FUNCTION_BLOCK SIMULATE
  {SET_ATTRIBUTE(OpcUa, SERVICE)}
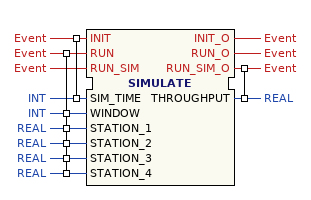
  EVENT_INPUT
    INIT WITH SIM_TIME;
    RUN WITH WINDOW, STATION_1, STATION_2, STATION_3, STATION_4; {SET_ATTRIBUTE(OpcUa, Method)}
    RUN_SIM; {SET_ATTRIBUTE(OpcUa, Method)}
  END_EVENT
  EVENT_OUTPUT
    INIT_O;
    RUN_O;
    RUN_SIM_O WITH THROUGHPUT;
  END_EVENT
  VAR_INPUT
    SIM_TIME : INT; {SET_ATTRIBUTE(OpcUa, Variable.RUN)}
    WINDOW : INT; {SET_ATTRIBUTE(OpcUa, Constant.RUN)}
    STATION_1 : REAL; {SET_ATTRIBUTE(OpcUa, Variable.RUN)}
    STATION_2 : REAL; {SET_ATTRIBUTE(OpcUa, Constant.RUN)}
    STATION_3 : REAL; {SET_ATTRIBUTE(OpcUa, Variable.RUN)}
    STATION_4 : REAL; {SET_ATTRIBUTE(OpcUa, Variable.RUN)}
  END_VAR
  VAR_OUTPUT
    THROUGHPUT : REAL; {SET_ATTRIBUTE(OpcUa, Variable.RUN)}
  END_VAR
END_FUNCTION_BLOCK
